{attribute 'linkalways'} 
{attribute 'no_explicit_call' := 'This FB is a CLASS and must be accessed using methods or properties'}
{attribute 'enable_dynamic_creation'}
FUNCTION_BLOCK FINAL OR_WORD EXTENDS Node
VAR
	in1 : _WORD(0);
	in2 : _WORD(0);
	out : _WORD(0);
END_VAR

METHOD PUBLIC Clone : I_Node
VAR
	pNode : POINTER TO OR_WORD;
END_VAR
pNode := __NEW(OR_WORD);
Clone := pNode^;
END_METHOD

METHOD FB_init : BOOL
VAR_INPUT
	bInitRetains : BOOL; // if TRUE, the retain variables are initialized (warm start / cold start)
	bInCopyCode : BOOL;  // if TRUE, the instance afterwards gets moved into the copy code (online change)
END_VAR
AddInput('in1',THIS^.in1);
AddInput('in2',THIS^.in2);
AddOutput('out', THIS^.out);
END_METHOD

METHOD PROTECTED OnExecute
VAR
END_VAR
out.Value := in1.Value OR in2.Value;
END_METHOD

END_FUNCTION_BLOCK

(* stored: Version 1.1.0.1, ProductVersion 3.1.4024.15
   POU OR_WORD: Id {c434fab8-3af4-4c27-9369-c8b6d0bd3851}, SpecialFunc None
   Folder Constructor: Id {9b3397d8-fc18-4198-8f1d-3f09c657923a}
   Method Clone: Id {a30cde7f-a76b-4a1e-9b30-7526f1aa8166}
   Method FB_init: Id {98f2b66f-0cf6-40e5-beb4-fed7d8b77a1c}
   Method OnExecute: Id {1c2d4d02-14a3-433c-9198-efb507e895f4} *)
